{attribute 'linkalways'} 
{attribute 'no_explicit_call' := 'This FB is a CLASS and must be accessed using methods or properties'}
{attribute 'enable_dynamic_creation'}
FUNCTION_BLOCK InvalidKeyDeserializationError EXTENDS Error
VAR
END_VAR

PROPERTY PUBLIC ErrorType : T_MAXSTRING
GET
ErrorType := 'INVALID_KEY_DESERIALIZATION_ERROR';
END_GET
END_PROPERTY

PROPERTY PUBLIC Message : T_MAXSTRING
GET
Message := 'Deserialization Failed, Key Cannot Be Empty';
END_GET
END_PROPERTY

END_FUNCTION_BLOCK

(* stored: Version 1.1.0.1, ProductVersion 3.1.4024.12
   POU InvalidKeyDeserializationError: Id {ed4d35f2-3487-0634-1035-11dc6206c2b9}, SpecialFunc None
   Property ErrorType: Id {65c56360-2817-0b6e-3d22-fb7371a45774}
   Get Get: Id {0f8392ac-83b6-084b-0cd6-136266b8055e}
   Property Message: Id {d5dd3561-0af0-0d84-3772-23a9a0d3af58}
   Get Get: Id {03a096d0-19da-0150-0d40-aac445117cac} *)
